{attribute 'GeneratedUsingTerminal: EK1122-0000-0018'}
{attribute addProperty BoxType "EK1122-0000-0018"}
{attribute addProperty Id "Beckhoff_EPP1xxxsub_EK1100EK1100_1FC0878B2A_0001_EPP1004_0061_0016EPP1004_D135F8DB8A_0002_EPP1008_0001_0016EPP1008_78E8D3DD12A_0003_EPP1008_0001_0017EPP1008_78E8D3DD12A_0004_EPP1008_0002_0016EPP1008_78E8D3DD12A_0005_EPP1008_0002_0017EPP1008_78E8D3DD12A_0006_EPP1008_0022_0016EPP1008_78E8D3DD12A_0007_EPP1018_0001_0016EPP1018_78E8D3DD12A_0008_EPP1018_0001_0017EPP1018_78E8D3DD12A_0009_EPP1018_0002_0016EPP1018_78E8D3DD12A_0010_EPP1018_0002_0017EPP1018_78E8D3DD12A_0011_EPP1111_0000_0016EPP1111_837A6B0314A_0012_EPP1111_0000_0017EPP1111_837A6B0314A_0013_EPP1111_0000_0018EPP1111_837A6B0314A_0014_EPP1258_0001_0016EPP1258_58F475DD56A_0015_EPP1258_0001_0017EPP1258_58F475DD56A_0016_EPP1258_0002_0016EPP1258_58F475DD56A_0017_EPP1258_0002_0017EPP1258_58F475DD56A_0018_EPP1321_0060_0016A_0018_EPP1321_0060_0016_F908F4F3378"}
{attribute addProperty CRC "1590345529"}
{attribute addProperty Size "762"}
TYPE Beckhoff_EPP1xxxEK1122_5ECABF39 EXTENDS EK1122_1FC0878B :
STRUCT
	{attribute addProperty Name "Beckhoff_EPP1xxxsub_EK1100"}
	{attribute addProperty PreviousPort "Beckhoff EPP1xxxEK1122 : D"}
	Beckhoff_EPP1xxxsub_EK1100 : EK1100_1FC0878B;
	{attribute addProperty Name "A_0001_EPP1004_0061_0016"}
	{attribute addProperty PreviousPort "Beckhoff EPP1xxxsub EK1100 : C"}
	A_0001_EPP1004_0061_0016 : EPP1004_D135F8DB;
	{attribute addProperty Name "A_0002_EPP1008_0001_0016"}
	{attribute addProperty PreviousPort "A_0001(EPP1004-0061-0016) : B"}
	A_0002_EPP1008_0001_0016 : EPP1008_78E8D3DD;
	{attribute addProperty Name "A_0003_EPP1008_0001_0017"}
	{attribute addProperty PreviousPort "A_0002(EPP1008-0001-0016) : B"}
	A_0003_EPP1008_0001_0017 : EPP1008_78E8D3DD;
	{attribute addProperty Name "A_0004_EPP1008_0002_0016"}
	{attribute addProperty PreviousPort "A_0003(EPP1008-0001-0017) : B"}
	A_0004_EPP1008_0002_0016 : EPP1008_78E8D3DD;
	{attribute addProperty Name "A_0005_EPP1008_0002_0017"}
	{attribute addProperty PreviousPort "A_0004(EPP1008-0002-0016) : B"}
	A_0005_EPP1008_0002_0017 : EPP1008_78E8D3DD;
	{attribute addProperty Name "A_0006_EPP1008_0022_0016"}
	{attribute addProperty PreviousPort "A_0005(EPP1008-0002-0017) : B"}
	A_0006_EPP1008_0022_0016 : EPP1008_78E8D3DD;
	{attribute addProperty Name "A_0007_EPP1018_0001_0016"}
	{attribute addProperty PreviousPort "A_0006(EPP1008-0022-0016) : B"}
	A_0007_EPP1018_0001_0016 : EPP1018_78E8D3DD;
	{attribute addProperty Name "A_0008_EPP1018_0001_0017"}
	{attribute addProperty PreviousPort "A_0007(EPP1018-0001-0016) : B"}
	A_0008_EPP1018_0001_0017 : EPP1018_78E8D3DD;
	{attribute addProperty Name "A_0009_EPP1018_0002_0016"}
	{attribute addProperty PreviousPort "A_0008(EPP1018-0001-0017) : B"}
	A_0009_EPP1018_0002_0016 : EPP1018_78E8D3DD;
	{attribute addProperty Name "A_0010_EPP1018_0002_0017"}
	{attribute addProperty PreviousPort "A_0009(EPP1018-0002-0016) : B"}
	A_0010_EPP1018_0002_0017 : EPP1018_78E8D3DD;
	{attribute addProperty Name "A_0011_EPP1111_0000_0016"}
	{attribute addProperty PreviousPort "A_0010(EPP1018-0002-0017) : B"}
	A_0011_EPP1111_0000_0016 : EPP1111_837A6B03;
	{attribute addProperty Name "A_0012_EPP1111_0000_0017"}
	{attribute addProperty PreviousPort "A_0011(EPP1111-0000-0016) : B"}
	A_0012_EPP1111_0000_0017 : EPP1111_837A6B03;
	{attribute addProperty Name "A_0013_EPP1111_0000_0018"}
	{attribute addProperty PreviousPort "A_0012(EPP1111-0000-0017) : B"}
	A_0013_EPP1111_0000_0018 : EPP1111_837A6B03;
	{attribute addProperty Name "A_0014_EPP1258_0001_0016"}
	{attribute addProperty PreviousPort "A_0013(EPP1111-0000-0018) : B"}
	A_0014_EPP1258_0001_0016 : EPP1258_58F475DD;
	{attribute addProperty Name "A_0015_EPP1258_0001_0017"}
	{attribute addProperty PreviousPort "A_0014(EPP1258-0001-0016) : B"}
	A_0015_EPP1258_0001_0017 : EPP1258_58F475DD;
	{attribute addProperty Name "A_0016_EPP1258_0002_0016"}
	{attribute addProperty PreviousPort "A_0015(EPP1258-0001-0017) : B"}
	A_0016_EPP1258_0002_0016 : EPP1258_58F475DD;
	{attribute addProperty Name "A_0017_EPP1258_0002_0017"}
	{attribute addProperty PreviousPort "A_0016(EPP1258-0002-0016) : B"}
	A_0017_EPP1258_0002_0017 : EPP1258_58F475DD;
	{attribute addProperty Name "A_0018_EPP1321_0060_0016"}
	{attribute addProperty PreviousPort "A_0017(EPP1258-0002-0017) : B"}
	A_0018_EPP1321_0060_0016 : A_0018_EPP1321_0060_0016_F908F4F3;
END_STRUCT
END_TYPE

(* stored: Version 1.2.0.0, ProductVersion 3.1.4024.9
   DUT Beckhoff_EPP1xxxEK1122_5ECABF39: Id {a5ba806f-3136-419c-bd27-cfbed496e3da} *)
